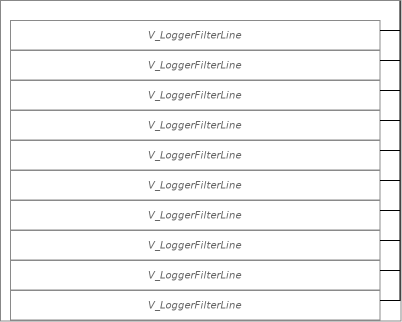
VISUALIZATION V_LoggerFilterList  // 402x322
VAR_IN_OUT
  IOfbLogger : FB_Logger;
	IOszFilterTxt : STRING(80);
END_VAR
    Line (400,300) (400,0)
    Frame (10,20 370x30)
        shows V_LoggerFilterLine(IOszTxtActual := IOszFilterTxt, IOszTxtLine := IOfbLogger.anvszVisuFilter[1])
    Frame (10,50 370x30)
        shows V_LoggerFilterLine(IOszTxtActual := IOszFilterTxt, IOszTxtLine := IOfbLogger.anvszVisuFilter[2])
    Frame (10,80 370x30)
        shows V_LoggerFilterLine(IOszTxtActual := IOszFilterTxt, IOszTxtLine := IOfbLogger.anvszVisuFilter[3])
    Frame (10,110 370x30)
        shows V_LoggerFilterLine(IOszTxtActual := IOszFilterTxt, IOszTxtLine := IOfbLogger.anvszVisuFilter[4])
    Frame (10,140 370x30)
        shows V_LoggerFilterLine(IOszTxtActual := IOszFilterTxt, IOszTxtLine := IOfbLogger.anvszVisuFilter[5])
    Line (380,30) (400,30)
    Line (380,60) (400,60)
    Line (380,90) (400,90)
    Line (380,120) (400,120)
    Line (380,150) (400,150)
    Frame (10,170 370x30)
        shows V_LoggerFilterLine(IOszTxtActual := IOszFilterTxt, IOszTxtLine := IOfbLogger.anvszVisuFilter[6])
    Frame (10,200 370x30)
        shows V_LoggerFilterLine(IOszTxtActual := IOszFilterTxt, IOszTxtLine := IOfbLogger.anvszVisuFilter[7])
    Frame (10,230 370x30)
        shows V_LoggerFilterLine(IOszTxtActual := IOszFilterTxt, IOszTxtLine := IOfbLogger.anvszVisuFilter[8])
    Frame (10,260 370x30)
        shows V_LoggerFilterLine(IOszTxtActual := IOszFilterTxt, IOszTxtLine := IOfbLogger.anvszVisuFilter[9])
    Frame (10,290 370x30)
        shows V_LoggerFilterLine(IOszTxtActual := IOszFilterTxt, IOszTxtLine := IOfbLogger.anvszVisuFilter[10])
    Line (380,180) (400,180)
    Line (380,210) (400,210)
    Line (380,240) (400,240)
    Line (380,270) (400,270)
    Line (380,300) (400,300)
END_VISUALIZATION

(* stored: Version 1.1.0.1, ProductVersion 3.1.4018.10
   Visu V_LoggerFilterList: Id {27d81015-2a94-4486-a562-610dafe59586} *)
